PROGRAM MAIN
VAR
	fbReadADS_1		: FB_ReadADS;
	bStart			: BOOL;
	bReset			: BOOL;
	fbWriteADS_1	: FB_WriteADS;
	bStartWrite		: BOOL;
	bResetWrite		: BOOL;
	i				: INT;
END_VAR

actComunicacao();

FOR i := 0 TO 20 DO
	GVL_ADS.Array_INT_Test[i] := i*33;
END_FOR

ACTION actComunicacao:
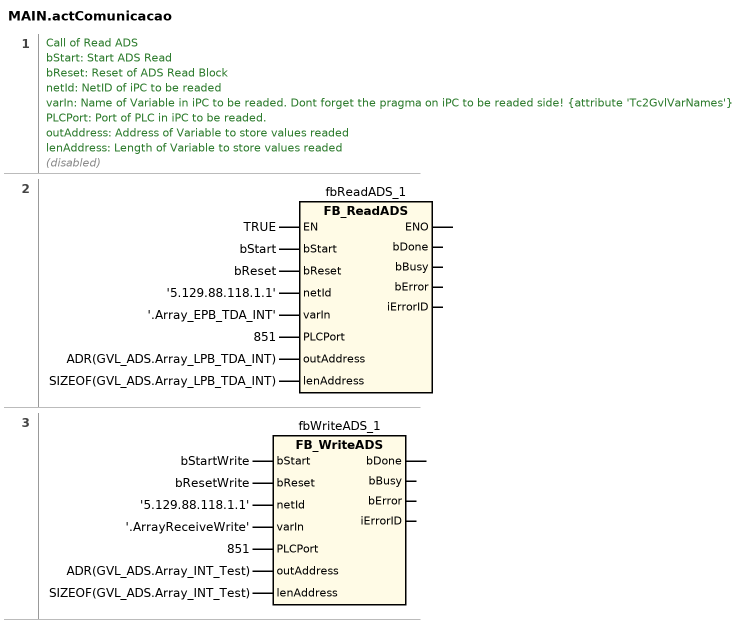
// NETWORK 1 (disabled)
// Call of Read ADS
// bStart: Start ADS Read
// bReset: Reset of ADS Read Block
// netId: NetID of iPC to be readed
// varIn: Name of Variable in iPC to be readed. Dont forget the pragma on iPC to be readed side! {attribute 'Tc2GvlVarNames'}
// PLCPort: Port of PLC in iPC to be readed.
// outAddress: Address of Variable to store values readed
// lenAddress: Length of Variable to store values readed

// NETWORK 2
fbReadADS_1(
    bStart := bStart,
    bReset := bReset,
    netId := '5.129.88.118.1.1',
    varIn := '.Array_EPB_TDA_INT',
    PLCPort := 851,
    outAddress := ADR(GVL_ADS.Array_LPB_TDA_INT),
    lenAddress := SIZEOF(GVL_ADS.Array_LPB_TDA_INT)); // FB_ReadADS

// NETWORK 3
fbWriteADS_1(
    bStart := bStartWrite,
    bReset := bResetWrite,
    netId := '5.129.88.118.1.1',
    varIn := '.ArrayReceiveWrite',
    PLCPort := 851,
    outAddress := ADR(GVL_ADS.Array_INT_Test),
    lenAddress := SIZEOF(GVL_ADS.Array_INT_Test)); // FB_WriteADS
END_ACTION

END_PROGRAM

(* stored: Version 1.1.0.1, ProductVersion 3.1.4024.12
   POU MAIN: Id {57912c50-efeb-4045-ad27-445a312d098c}, SpecialFunc None
   Action actComunicacao: Id {e157e37b-04a8-4e2f-b1a9-0b6e35d0a88c} *)
